{attribute 'GeneratedUsingTerminal: EL3773-0000-0021'}
{attribute addProperty BoxType "EL3773-0000-0021"}
{attribute addProperty Id "U1_SamplesAT %I*U1_Samples_2549228720"}
{attribute addProperty CRC "1101969407"}
{attribute addProperty Size "20"}
TYPE L1_Voltage_Samples_41AEB7FF EXTENDS TcoIo.InputBase_8311D824 : STRUCT
    {attribute addProperty Name "U1_Samples"}
    U1_Samples AT %I* : U1_Samples_25492287;
END_STRUCT
END_TYPE

(* stored: Version 1.2.0.0, ProductVersion 3.1.4024.11
   DUT L1_Voltage_Samples_41AEB7FF: Id {f17555da-12a7-03d4-039d-d40e8c5aca5f} *)
